Fanuc KAREL source: kt00504.KL

-- PROVISIONAL review KL for V770-1; original PC SHA256 76b736e0b3aa51b0eb7d747228f33324dfe690e1190c1794984f7433a0e8815a
-- Incomplete behavior may be omitted. Consult companion uncertainty JSON. Do not deploy.
PROGRAM KT00504
%NOLOCKGROUP
-- UNRESOLVED_DECL P1 type=000102
-- UNRESOLVED_DECL P2 type=000106
-- UNRESOLVED_DECL OUT type=000101
BEGIN
  -- UNRESOLVED_PC offsets 5-20; opcodes 2E,22,32,35
  -- UNRESOLVED_PC offsets 25-40; opcodes 2E,22,32,35
  -- UNRESOLVED_PC offsets 45-79; opcodes 49,7E,49,7E,60,4A
  -- UNRESOLVED_PC offsets 84-88; opcodes 7F
END KT00504
